FUNCTION ST08B_TO_BYTES (* this Function extracts the 8 BYTES from a 8-BYTE Struct *)
  (* Standard: 61499-1; Description: Copyright (c) 2024 HR Agrartechnik GmbH This program and the accompanying materials are made available under the terms of the Eclipse Public License 2.0 which is available at https://www.eclipse.org/legal/epl-2.0/ SPDX-License-Identifier: EPL-2.0 *)
  (* Version 1.0, 2024-02-22, Franz Höpfinger, HR Agrartechnik GmbH *)
  PACKAGE logiBUS::utils::conversion::str::forwarding;
  IMPORT eclipse4diac::core::TypeHash;
  IMPORT logiBUS::utils::conversion::types::ST08B;
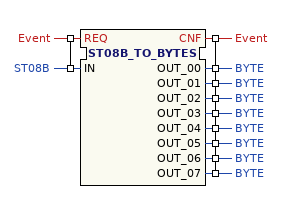
  EVENT_INPUT
    REQ WITH IN;
  END_EVENT
  EVENT_OUTPUT
    CNF WITH OUT_00, OUT_01, OUT_02, OUT_03, OUT_04, OUT_05, OUT_06, OUT_07;
  END_EVENT
  VAR_INPUT
    IN : logiBUS::utils::conversion::types::ST08B; (* ST08B Input *)
  END_VAR
  VAR_OUTPUT
    OUT_00 : BYTE; (* BYTE 00 *)
    OUT_01 : BYTE; (* BYTE 01 *)
    OUT_02 : BYTE; (* BYTE 02 *)
    OUT_03 : BYTE; (* BYTE 03 *)
    OUT_04 : BYTE; (* BYTE 04 *)
    OUT_05 : BYTE; (* BYTE 05 *)
    OUT_06 : BYTE; (* BYTE 06 *)
    OUT_07 : BYTE; (* BYTE 07 *)
  END_VAR
  BODY IN ST:
PACKAGE logiBUS::utils::conversion::str::forwarding;

IMPORT logiBUS::utils::conversion::types::ST08B;

(* this Function extracts the 8 BYTES from a 8-BYTE Struct *)
FUNCTION ST08B_TO_BYTES

VAR_INPUT
	IN : ST08B; // ST08B Input
END_VAR

VAR_OUTPUT
	OUT_00 : BYTE; // BYTE 00
	OUT_01 : BYTE; // BYTE 01
	OUT_02 : BYTE; // BYTE 02
	OUT_03 : BYTE; // BYTE 03
	OUT_04 : BYTE; // BYTE 04
	OUT_05 : BYTE; // BYTE 05
	OUT_06 : BYTE; // BYTE 06
	OUT_07 : BYTE; // BYTE 07
END_VAR

OUT_00 := IN.B_00;
OUT_01 := IN.B_01;
OUT_02 := IN.B_02;
OUT_03 := IN.B_03;
OUT_04 := IN.B_04;
OUT_05 := IN.B_05;
OUT_06 := IN.B_06;
OUT_07 := IN.B_07;

END_FUNCTION
  END_BODY
END_FUNCTION
